      A     #i_TRS2_EXT_Inputs.Request_Stop; // IF External stop Request
      O     #s_TRS2_ST_PEC_Block; // OR PEC blockage
      O     #o_TRS2_ST_PPI_Err; // OR PPI error
      O     #s_TRS2_ST_LMS_ASI_Not_Pr; // OR LMS ASI not present
      O     #s_TRS2_ST_LMS_ASI_Error; // OR LMS ASI Error
      O     #s_TRS2_ST_LMS_Not_Health; // OR LMS not healthy
      O     #s_TRS2_ST_PEC_Missings; // OR PEC missing
      O     #s_TRS2_ST_LMS_Not_Auto; // OR in automatic mode
      O     #s_Req_Stop_TRS2; // OR request to stop TRS 2 due to error of VBS or SWS
      =     #s_TRS2_Req_Stop; // Request Stop

// Request Halt to the section
      A     #i_Ext_Req_Dis_Send;
      O     #s_Halt_TRS2_Gap_Not_Clr; // Halt TRS2 when the gap clear area is not clear and the divert section is not running
      O     #s_Halt_TRS2_Dir1;
      O     #s_Halt_TRS2_Dir2;
      O     #s_Halt_TRS2_Belt_NOK;
      O     #s_DecPoint_Wait_TRS2; // Settings at decision point are configured to halt the item in front of the vertibelt
      O     #i_TRS2_EXT_Inputs.Request_Halt; // IF External halt Request
      =     #s_TRS2_Req_Halt;

      CALL "FC_PLT_Clr_DB" (
           i_Enable_Clr             := #s_TRS2_ST_LMS_Not_Auto,
           i_DB_PLT_Num             := #t_DB_PLT_TRS2,
           i_DB_Event_Num           := #s_DB_Num_Event);

      CALL #s_TRS2_FB_EQP_Basic (
           i_ID_Section             := #i_TRS2_ID,
           i_Setting                := #i_TRS2_Setting.Basic,
           i_DB_PLT                 := #i_TRS2_DB_PLT,
           i_DB_PLT_DwnStr          := #i_TRS2_DB_PLT_Downstr,
           i_DB_Event               := "DB_Event_Section",
           i_CFG_Conveyor_Speed     := #i_TRS2_CFG_Conv_Speed,
           i_CFG_Run_Out_Distance   := #i_TRS2_CFG_Run_Out_Dist,
           i_CFG_Minimum_Gap        := #i_CFG_TRS2_Minimum_Gap,
           i_CFG_Add_Gap_Stop       := #i_CFG_TRS2_Add_Gap_Stop,
           i_CFG_Minimum_H2H        := #i_CFG_TRS2_Minimum_H2H,
           i_CFG_Add_H2H_Stop       := #i_CFG_TRS2_Add_H2H_Stop,
           i_CFG_Cascade_Delay_Time := 300,
           i_CFG_Strt_Up_T_E_Save   := "DB_Setting".common.Start_Up_Time_E_Save,
           i_CFG_Run_Out_E_Save     := "DB_Setting".common.Run_Out_Time_E_Save,
           i_CFG_Stop_T_E_Save      := "DB_Setting".common.Stop_Time_E_Save,
           i_CFG_Disbl_E_Save       := "DB_Setting".common.Disable_Energy_Saving,
           i_CFG_Slave_Mode         := FALSE,
           i_CFG_Del_Window_Codes   := FALSE,
           i_PPI_Displacement       := 0,
           i_Dwnstr_PLT_Pos         := #s_TRS2_Int_Prog.PEC_Offset,
           i_Available_IO           := #i_TRS2_Available_IO,
           i_Safety_OK              := #i_Safety_OK,
           i_CMD_Enable             := #i_CMD_Enable,
           i_CMD_Start              := #i_CMD_Start,
           i_Ext_Req_Stop           := #s_TRS2_Req_Stop,
           i_Ext_Req_Halt           := #s_TRS2_Req_Halt,
           i_Ext_Req_Dis_Send       := #i_TRS2_EXT_Inputs.Request_Disable_Send,
           i_Ext_Req_Rst_ESave      := #i_TRS2_EXT_Inputs.Request_Reset_EnergySave,
           i_OS_Direction_Change    := FALSE,
           o_External               := #o_TRS2_EXT_Outputs,
           o_Motor_Run              := #s_TRS2_Int_Prog.Motor_Run,
           o_ST_Items               := #o_TRS2_ST_Items,
           o_ST_Running             := #o_TRS2_ST_Running,
           o_ST_Started             := #o_TRS2_ST_Started,
           o_ST_Request_Halt        := #o_TRS2_ST_Req_Halt,
           o_ST_Request_Stop        := #o_TRS2_ST_Req_Stop,
           o_Ready_To_Restart       := #s_TRS2_Ready_Restart);

      CALL #s_TRS2_FB_TRK_Track (
           i_Trigger_Send_Stat      := #i_CMD_Send_Stat,
           i_CMD_Reset              := #i_CMD_Reset,
           i_DB_PLT                 := #i_TRS2_DB_PLT,
           i_Event_DB               := "DB_Event_Section",
           i_Position_PEC_Update    := #s_TRS2_Int_Prog.PEC_Offset,
           i_LPOS                   := #s_TRS2_Int_Prog.LPOS,
           i_Setting                := #i_TRS2_Setting.Tracking,
           i_CFG_Clear_Double_Data  := FALSE,
           i_Length_Dif_Accepted    := 0,
           i_CFG_Num_Missing_Error  := 3,
           i_CFG_Upd_Perf_WN_Level  := 80,
           i_CFG_Weighing_Factor    := 10,
           i_CFG_Default_Record     := #i_CFG_Default_Record,
           i_OS_Direction_Change    := FALSE,
           o_ST_PEC_Miss            := #s_TRS2_ST_PEC_Missings,
           o_ST_PEC_BadTrack        := #o_TRS2_ST_Bad_Update);

      CALL #s_TRS2_FB_HW_MTR_LMS (
           i_CMD_Send_Stat          := #i_CMD_Send_Stat,
           i_Event_DB               := "DB_Event_Section",
           i_Available_IO           := #i_TRS2_Available_IO,
           i_Quick_Stop             := FALSE,
           i_LMS_NotPrsnt           := #i_TRS2_IO_LMS_NotPrsnt,
           i_LMS_Error              := #i_TRS2_IO_LMS_Error,
           i_IO_LMS_Auto            := #i_TRS2_IO_LMS_Auto,
           i_IO_LMS_Healthy         := #i_TRS2_IO_LMS_Healthy,
           i_CMD_Reset              := #i_CMD_Reset,
           i_CMD_Req_Motor_Forward  := #s_TRS2_Int_Prog.Motor_Run,
           o_IO_MTR_Fwd             := #o_TRS2_IO_MTR_Fwd,
           o_IO_MTR_Rev             := #o_TRS2_IO_MTR_Rev,
           o_IO_MTR_Dis_Quick_Stop  := #o_TRS2_IO_Disable_QS,
           o_ST_ASI_NotPrsnt        := #s_TRS2_ST_LMS_ASI_Not_Pr,
           o_ST_ASI_Err             := #s_TRS2_ST_LMS_ASI_Error,
           o_ST_LMS_Not_Auto        := #s_TRS2_ST_LMS_Not_Auto,
           o_ST_LMS_Not_Hthy        := #s_TRS2_ST_LMS_Not_Health);

      CALL #s_TRS2_Window_Generator (
           i_DB_PLT_Most_DwnStr     := #i_TRS2_DB_PLT,
           i_DB_PLT_Most_UpStr      := #i_TRS2_DB_PLT,
           i_DB_Reservation         := #i_DB_Res_TRS2,
           i_DB_Event               := "DB_Event_Zone",
           i_CFG_Window_Length      := #s_Calc_H2H_Length_VBS1,
           i_CFG_In_Flow_Function   := FALSE,
           i_Section_Run_Reverse    := FALSE);

      CALL #s_FB_DAT_TRS2 (
           i_ID_Section             := #i_TRS2_ID,
           i_DB_Event               := "DB_Event_Section",
           i_PLC_FIFO_DB            := "DB_Send_FIFO",
           i_PLC_Log_FIFO_DB        := "DB_LOG_Event_FIFO",
           i_Degraded_Mode          := "M_Comm_Degraded",
           i_CFG_BPI_Log_Level      := "DB_Setting".common.External_Log_Level,
           i_CFG_PLC_Log_Level      := "DB_Setting".common.Internal_Log_Level,
           i_CFG_PLC_Log_SAC_Mesgs  := FALSE,
           i_CFG_PLC_LOG_BPI_Stat   := FALSE);

NETWORK
TITLE =UA: Right sorter section (TRS3)

      NOP   0;
// Induct from section upstream of TRS3 onto TRS3 is only used when flow A is active
      A     #s_Flow_A;
      JCN   UA01;

      CALL #s_TRS3_FB_Induct (
           i_Setting                := #i_Setting.Induct_Upstr_TRS3_Sett,
           i_DB_PLT                 := #i_TRS3_Ups_Induct_DB_PLT,
           i_DB_PLT_Merge           := #i_TRS3_DB_PLT,
           i_DB_Reservation         := #i_DB_Res_TRS3,
           i_DB_Event               := "DB_Event_Zone",
           i_CFG_PEC_Offset         := #s_TRS3_Int_Prog.PEC_Offset,
           i_CFG_Search_Window      := 0,
           i_CFG_Gap_Length         := 20,
           i_CFG_Induct_Number_FWD  := 2,
           i_CFG_Run_Out_Dist_Gap   := #i_TRS3_Ups_Run_Out_Dist);

// When using the induct block connect the induct PLT DB inbetween TRS3 and it's upstream section
      OPN   #i_TRS3_DB_PLT;
      L     0; //#s_Upst_TRS3_IND_DB_PLT
      T     DBW    6;

      OPN   #i_TRS3_DB_PLT_Upstr;
      L     #s_Upst_TRS3_IND_DB_PLT;
      T     DBW    8;

      OPN   #i_TRS3_Ups_Induct_DB_PLT;
      L     #s_TRS3_DB_PLT_Upstream;
      T     DBW    6;
      L     #t_DB_PLT_TRS3;
      T     DBW    8;
      JU    UA02;

// When not using the induct block connect TRS3 direct to it's upstream section.
UA01: OPN   #i_TRS3_DB_PLT;
      L     #s_TRS3_DB_PLT_Upstream;
      T     DBW    6;

      OPN   #i_TRS3_DB_PLT_Upstr;
      L     #t_DB_PLT_TRS3;
      T     DBW    8;

UA02: NOP   0;

      CALL "FC_Calc_H2H_Distance" (
           i_CFG_Conveyor_Speed     := #i_TRS3_CFG_Conv_Speed,
           i_CFG_Capacity           := 1200,
           i_CFG_Minimum_Capacity   := 1200,
           i_CFG_Maximum_Capacity   := 1200,
           o_H2H_Length             := #s_Calc_H2H_Length_VBS2,
           o_Current_Capacity       := #o_Capacity_VBS2,
           o_ST_Capacity_2Low       := #t_Not_Used_Bool,
           o_ST_Capacity_2High      := #t_Not_Used_Bool,
           o_ST_CalcH2H_Disable     := #t_Not_Used_Bool);

      CALL #s_TRS3_FB_EQP_PEC (
           i_Setting                := #i_TRS3_Setting.PEC_1D,
           i_DB_PLT                 := #i_TRS3_DB_PLT,
           i_DB_Event               := "DB_Event_Section",
           i_Dwnstr_PLT_Pos         := 0,
           i_CFG_Blockage_Length    := 300,
           i_CFG_Delay_On_Filter    := 0,
           i_CFG_Delay_Off_Filter   := 20,
           i_CFG_Min_Product_Length := 0,
           i_CFG_Preset_PEC_Latch   := #s_TRS3_ST_LMS_Not_Auto,
           i_CFG_Track_Present      := TRUE,
           i_CFG_Reset_Block_PEC_Oc := FALSE,
           i_IO_NOT_PEC             := #i_TRS3_IO_NOT_PEC,
           i_Eqp_Available_IO       := #i_TRS3_Available_IO,
           i_CMD_Reset              := #i_CMD_Reset,
           o_LPOS                   := #s_TRS3_Int_Prog.LPOS,
           o_PEC_Position           := #s_TRS3_Int_Prog.PEC_Offset,
           o_ST_PEC_Blk             := #s_TRS3_ST_PEC_Block);

      CALL #s_TRS3_FB_EQP_PPI (
           i_CFG_PPI_Resolution     := 50,
           i_CFG_Time_Out_Error     := 300,
           i_DB_PLT                 := #i_TRS3_DB_PLT,
           i_IO_PPI                 := #i_TRS3_IO_PPI,
           i_CMD_Reset              := #i_CMD_Reset,
           o_PPI_Displacement_mm    := #s_TRS3_Int_Prog.PPI_Displacement,
           o_ST_PPI_Err             := #o_TRS3_ST_PPI_Err);

// Request stop for basic equipment
      A     #s_VBS2_ST_Not_Automatic;
      O     #s_SWS_VBS2_Gap_NotClr;
      O     #s_SWS2_ST_Move_Time_Out;
      O     #s_VBS2_ST_Not_Healthy;
      O     #s_VBS2_ST_ASI_Not_Prsnt;
      O     #s_VBS2_ST_ASI_Error;
      O     #s_SWS2_ST_ASI_Not_Presnt;
      O     #s_SWS2_ST_ASI_Error;
      O     #s_SWS2_ST_Err_PS_Double;
      O     #s_TRS1_ST_PEC_Block_1;
      =     #s_Req_Stop_TRS3;

      A     #i_TRS3_EXT_Inputs.Request_Stop; // IF External stop Request
      O     #s_TRS3_ST_PEC_Block; // OR PEC blockage
      O     #o_TRS3_ST_PPI_Err; // OR PPI error
      O     #s_TRS3_ST_LMS_ASI_Not_Pr; // OR LMS ASI not present
      O     #s_TRS3_ST_LMS_ASI_Error; // OR LMS ASI Error
      O     #s_TRS3_ST_LMS_Not_Health; // OR LMS not healthy
      O     #s_TRS3_ST_PEC_Missings; // OR PEC missing
      O     #s_TRS3_ST_LMS_Not_Auto; // OR in automatic mode
      O     #s_Req_Stop_TRS3;
      =     #s_TRS3_Req_Stop; // Request Stop

// Request Halt to the section
      A     #i_Ext_Req_Dis_Send;
      O     #s_Halt_TRS3_Gap_Not_CLR; // Halt TRS3 when the gap clear area is not clear and the divert section is not running
      O     #s_Halt_TRS3_Dir1;
      O     #s_Halt_TRS3_Dir2;
      O     #s_Halt_TRS3_Belt_NOK;
      O     #s_DecPoint_Wait_TRS3; // Settings at decision point are configured to halt the item in front of the vertibelt
      O     #i_TRS3_EXT_Inputs.Request_Halt; // IF External halt Request
      =     #s_TRS3_Req_Halt;

      CALL "FC_PLT_Clr_DB" (
           i_Enable_Clr             := #s_TRS3_ST_LMS_Not_Auto,
           i_DB_PLT_Num             := #t_DB_PLT_TRS3,
           i_DB_Event_Num           := #s_DB_Num_Event);

      CALL #s_TRS3_FB_EQP_Basic (
           i_ID_Section             := #i_TRS3_ID,
           i_Setting                := #i_TRS3_Setting.Basic,
           i_DB_PLT                 := #i_TRS3_DB_PLT,
           i_DB_PLT_DwnStr          := #i_TRS3_DB_PLT_Downstream,
           i_DB_Event               := "DB_Event_Section",
           i_CFG_Conveyor_Speed     := #i_TRS3_CFG_Conv_Speed,
           i_CFG_Run_Out_Distance   := #i_TRS3_CFG_Run_Out_Dist,
           i_CFG_Minimum_Gap        := #i_CFG_TRS3_Minimum_Gap,
           i_CFG_Add_Gap_Stop       := #i_CFG_TRS3_Add_Gap_Stop,
           i_CFG_Minimum_H2H        := #i_CFG_TRS3_Minimum_H2H,
           i_CFG_Add_H2H_Stop       := #i_CFG_TRS3_Add_H2H_Stop,
           i_CFG_Cascade_Delay_Time := 300,
           i_CFG_Strt_Up_T_E_Save   := "DB_Setting".common.Start_Up_Time_E_Save,
           i_CFG_Run_Out_E_Save     := "DB_Setting".common.Run_Out_Time_E_Save,
           i_CFG_Stop_T_E_Save      := "DB_Setting".common.Stop_Time_E_Save,
           i_CFG_Disbl_E_Save       := "DB_Setting".common.Disable_Energy_Saving,
           i_CFG_Slave_Mode         := FALSE,
           i_CFG_Del_Window_Codes   := FALSE,
           i_PPI_Displacement       := 0,
           i_Dwnstr_PLT_Pos         := #s_TRS3_Int_Prog.PEC_Offset,
           i_Available_IO           := #i_TRS3_Available_IO,
           i_Safety_OK              := #i_Safety_OK,
           i_CMD_Enable             := #i_CMD_Enable,
           i_CMD_Start              := #i_CMD_Start,
           i_Ext_Req_Stop           := #s_TRS3_Req_Stop,
           i_Ext_Req_Halt           := #s_TRS3_Req_Halt,
           i_Ext_Req_Dis_Send       := #i_TRS3_EXT_Inputs.Request_Disable_Send,
           i_Ext_Req_Rst_ESave      := #i_TRS3_EXT_Inputs.Request_Reset_EnergySave,
           i_OS_Direction_Change    := FALSE,
           o_External               := #o_TRS3_EXT_Outputs,
           o_Motor_Run              := #s_TRS3_Int_Prog.Motor_Run,
           o_ST_Items               := #o_TRS3_ST_Items,
           o_ST_Running             := #o_TRS3_ST_Running,
           o_ST_Started             := #o_TRS3_ST_Started,
           o_ST_Request_Halt        := #o_TRS3_ST_Req_Halt,
           o_ST_Request_Stop        := #o_TRS3_ST_Req_Stop,
           o_Ready_To_Restart       := #s_TRS3_Ready_Restart);

      CALL #s_TRS3_FB_TRK_Track (
           i_Trigger_Send_Stat      := #i_CMD_Send_Stat,
           i_CMD_Reset              := #i_CMD_Reset,
           i_DB_PLT                 := #i_TRS3_DB_PLT,
           i_Event_DB               := "DB_Event_Section",
           i_Position_PEC_Update    := #s_TRS3_Int_Prog.PEC_Offset,
           i_LPOS                   := #s_TRS3_Int_Prog.LPOS,
           i_Setting                := #i_TRS3_Setting.Tracking,
           i_CFG_Clear_Double_Data  := FALSE,
           i_Length_Dif_Accepted    := 0,
           i_CFG_Num_Missing_Error  := 3,
           i_CFG_Upd_Perf_WN_Level  := 80,
           i_CFG_Weighing_Factor    := 10,
           i_CFG_Default_Record     := #i_CFG_Default_Record,
           i_OS_Direction_Change    := FALSE,
           o_ST_PEC_Miss            := #s_TRS3_ST_PEC_Missings,
           o_ST_PEC_BadTrack        := #o_TRS3_ST_Bad_Update);

      CALL #s_TRS3_FB_HW_MTR_LMS (
           i_CMD_Send_Stat          := #i_CMD_Send_Stat,
           i_Event_DB               := "DB_Event_Section",
           i_Available_IO           := #i_TRS3_Available_IO,
           i_Quick_Stop             := FALSE,
           i_LMS_NotPrsnt           := #i_TRS3_IO_LMS_NotPrsnt,
           i_LMS_Error              := #i_TRS3_IO_LMS_Error,
           i_IO_LMS_Auto            := #i_TRS3_IO_LMS_Auto,
           i_IO_LMS_Healthy         := #i_TRS3_IO_LMS_Healthy,
           i_CMD_Reset              := #i_CMD_Reset,
           i_CMD_Req_Motor_Forward  := #s_TRS3_Int_Prog.Motor_Run,
           o_IO_MTR_Fwd             := #o_TRS3_IO_MTR_Fwd,
           o_IO_MTR_Rev             := #o_TRS3_IO_MTR_Rev,
           o_IO_MTR_Dis_Quick_Stop  := #o_TRS3_IO_Disable_QS,
           o_ST_ASI_NotPrsnt        := #s_TRS3_ST_LMS_ASI_Not_Pr,
           o_ST_ASI_Err             := #s_TRS3_ST_LMS_ASI_Error,
           o_ST_LMS_Not_Auto        := #s_TRS3_ST_LMS_Not_Auto,
           o_ST_LMS_Not_Hthy        := #s_TRS3_ST_LMS_Not_Health);

      CALL #s_TRS3_Window_Generator (
           i_DB_PLT_Most_DwnStr     := #i_TRS3_DB_PLT,
           i_DB_PLT_Most_UpStr      := #i_TRS3_DB_PLT,
           i_DB_Reservation         := #i_DB_Res_TRS3,
           i_DB_Event               := "DB_Event_Zone",
           i_CFG_Window_Length      := #s_Calc_H2H_Length_VBS2,
           i_CFG_In_Flow_Function   := FALSE,
           i_Section_Run_Reverse    := FALSE);

      CALL #s_FB_DAT_TRS3 (
           i_ID_Section             := #i_TRS3_ID,
           i_DB_Event               := "DB_Event_Section",
           i_PLC_FIFO_DB            := "DB_Send_FIFO",
           i_PLC_Log_FIFO_DB        := "DB_LOG_Event_FIFO",
           i_Degraded_Mode          := "M_Comm_Degraded",
           i_CFG_BPI_Log_Level      := "DB_Setting".common.External_Log_Level,
           i_CFG_PLC_Log_Level      := "DB_Setting".common.Internal_Log_Level,
           i_CFG_PLC_Log_SAC_Mesgs  := FALSE,
           i_CFG_PLC_LOG_BPI_Stat   := FALSE);

NETWORK
TITLE =VA: Data Layer of VBZ
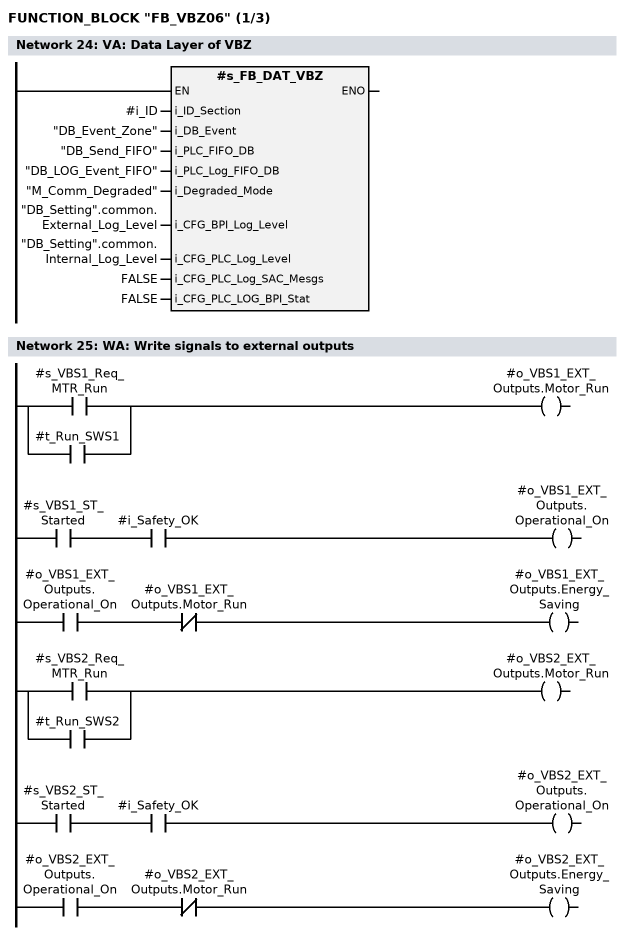

      CALL #s_FB_DAT_VBZ (
           i_ID_Section             := #i_ID,
           i_DB_Event               := "DB_Event_Zone",
           i_PLC_FIFO_DB            := "DB_Send_FIFO",
           i_PLC_Log_FIFO_DB        := "DB_LOG_Event_FIFO",
           i_Degraded_Mode          := "M_Comm_Degraded",
           i_CFG_BPI_Log_Level      := "DB_Setting".common.External_Log_Level,
           i_CFG_PLC_Log_Level      := "DB_Setting".common.Internal_Log_Level,
           i_CFG_PLC_Log_SAC_Mesgs  := FALSE,
           i_CFG_PLC_LOG_BPI_Stat   := FALSE);

NETWORK
TITLE =WA: Write signals to external outputs

      NOP   0;
// Signals for VBS 1
      A     #s_VBS1_Req_MTR_Run;
      O     #t_Run_SWS1;
      =     #o_VBS1_EXT_Outputs.Motor_Run;

      A     #s_VBS1_ST_Started;
      A     #i_Safety_OK;
      =     #o_VBS1_EXT_Outputs.Operational_On;

      A     #o_VBS1_EXT_Outputs.Operational_On;
      AN    #o_VBS1_EXT_Outputs.Motor_Run;
      =     #o_VBS1_EXT_Outputs.Energy_Saving;

// Signals for VBS 2
      A     #s_VBS2_Req_MTR_Run;
      O     #t_Run_SWS2;
      =     #o_VBS2_EXT_Outputs.Motor_Run;

      A     #s_VBS2_ST_Started;
      A     #i_Safety_OK;
      =     #o_VBS2_EXT_Outputs.Operational_On;

      A     #o_VBS2_EXT_Outputs.Operational_On;
      AN    #o_VBS2_EXT_Outputs.Motor_Run;
      =     #o_VBS2_EXT_Outputs.Energy_Saving;
NETWORK
TITLE =XA: Write zone status
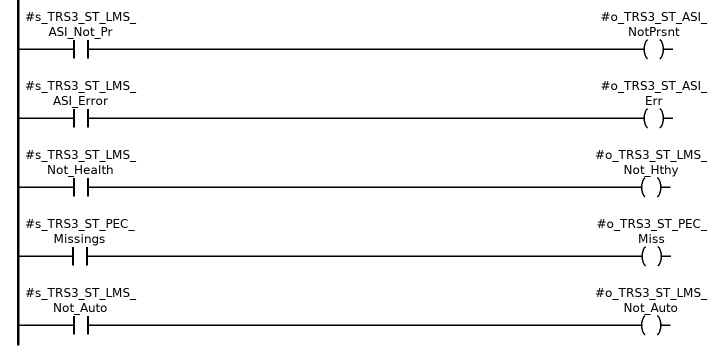

      A     #s_Flow_Straight;
      =     #o_ST_Fixed_Straight;

      A     #s_Flow_A;
      =     #o_ST_Fixed_Flow_A;

      A     #s_Flow_B;
      =     #o_ST_Fixed_Flow_B;

      A     #s_VBS1_ST_Started;
      AN    #s_VBS1_ST_Not_Automatic;
      AN    #s_VBS1_ST_Not_Healthy;
      AN    #s_VBS1_ST_ASI_Not_Prsnt;
      AN    #s_VBS1_ST_ASI_Error;
      =     #o_VBS1_ST_Started;

      A     #s_VBS2_ST_Started;
      AN    #s_VBS2_ST_Not_Automatic;
      AN    #s_VBS2_ST_Not_Healthy;
      AN    #s_VBS2_ST_ASI_Not_Prsnt;
      AN    #s_VBS2_ST_ASI_Error;
      =     #o_VBS2_ST_Started;

// Copy section statusses to outputs

      A     #s_VBS1_ST_ASI_Not_Prsnt;
      =     #o_VBS1_ST_ASI_NotPrsnt;

      A     #s_VBS1_ST_ASI_Error;
      =     #o_VBS1_ST_ASI_Err;

      A     #s_VBS1_ST_Not_Automatic;
      =     #o_VBS1_ST_LMS_Not_Auto;

      A     #s_VBS1_ST_Not_Healthy;
      =     #o_VBS1_ST_LMS_Not_Hthy;

      A     #s_SWS1_ST_ASI_Not_Presnt;
      =     #o_SWS1_ST_ASI_NotPrsnt;

      A     #s_SWS1_ST_ASI_Error;
      =     #o_SWS1_ST_ASI_Error;

      A     #s_SWS1_ST_Not_Automatic;
      =     #o_SWS1_ST_Not_Automatic;

      A     #s_SWS1_ST_Not_Healthy;
      =     #o_SWS1_ST_Not_Healthy;

      A     #s_SWS1_ST_Move_Time_Out;
      =     #o_SWS1_ST_Move_Time_Out;

      A     #s_SWS1_ST_Err_PS_Double;
      =     #o_SWS1_ST_Err_PS_Double;

      A     #s_VBS2_ST_ASI_Not_Prsnt;
      =     #o_VBS2_ST_ASI_NotPrsnt;

      A     #s_VBS2_ST_ASI_Error;
      =     #o_VBS2_ST_ASI_Err;

      A     #s_VBS2_ST_Not_Automatic;
      =     #o_VBS2_ST_LMS_Not_Auto;

      A     #s_VBS2_ST_Not_Healthy;
      =     #o_VBS2_ST_LMS_Not_Hthy;

      A     #s_SWS2_ST_ASI_Not_Presnt;
      =     #o_SWS2_ST_ASI_NotPrsnt;

      A     #s_SWS2_ST_ASI_Error;
      =     #o_SWS2_ST_ASI_Error;

      A     #s_SWS2_ST_Not_Automatic;
      =     #o_SWS2_ST_Not_Automatic;

      A     #s_SWS2_ST_Not_Healthy;
      =     #o_SWS2_ST_Not_Healthy;

      A     #s_SWS2_ST_Move_Time_Out;
      =     #o_SWS2_ST_Move_Time_Out;

      A     #s_SWS2_ST_Err_PS_Double;
      =     #o_SWS2_ST_Err_PS_Double;

      A     #s_TRS1_ST_PEC_Block_1;
      =     #o_TRS1_ST_PEC_Blk;

      A     #s_TRS1_ST_PEC_Block_2;
      =     #o_TRS1_ST_PEC2_Blk;

      A     #s_TRS1_ST_LMS_ASI_Not_Pr;
      =     #o_TRS1_ST_ASI_NotPrsnt;

      A     #s_TRS1_ST_LMS_ASI_Error;
      =     #o_TRS1_ST_ASI_Err;

      A     #s_TRS1_ST_LMS_Not_Health;
      =     #o_TRS1_ST_LMS_Not_Hthy;

      A     #s_TRS1_ST_PEC_Missings;
      =     #o_TRS1_ST_PEC_Miss;

      A     #s_TRS1_ST_LMS_Not_Auto;
      =     #o_TRS1_ST_LMS_Not_Auto;

      A     #s_TRS2_ST_PEC_Block;
      =     #o_TRS2_ST_PEC_Blk;

      A     #s_TRS2_ST_LMS_ASI_Not_Pr;
      =     #o_TRS2_ST_ASI_NotPrsnt;

      A     #s_TRS2_ST_LMS_ASI_Error;
      =     #o_TRS2_ST_ASI_Err;

      A     #s_TRS2_ST_LMS_Not_Health;
      =     #o_TRS2_ST_LMS_Not_Hthy;

      A     #s_TRS2_ST_PEC_Missings;
      =     #o_TRS2_ST_PEC_Miss;

      A     #s_TRS2_ST_LMS_Not_Auto;
      =     #o_TRS2_ST_LMS_Not_Auto;

      A     #s_TRS3_ST_PEC_Block;
      =     #o_TRS3_ST_PEC_Blk;

      A     #s_TRS3_ST_LMS_ASI_Not_Pr;
      =     #o_TRS3_ST_ASI_NotPrsnt;

      A     #s_TRS3_ST_LMS_ASI_Error;
      =     #o_TRS3_ST_ASI_Err;

      A     #s_TRS3_ST_LMS_Not_Health;
      =     #o_TRS3_ST_LMS_Not_Hthy;

      A     #s_TRS3_ST_PEC_Missings;
      =     #o_TRS3_ST_PEC_Miss;

      A     #s_TRS3_ST_LMS_Not_Auto;
      =     #o_TRS3_ST_LMS_Not_Auto;

NETWORK
TITLE =YA: Write zone status request signals
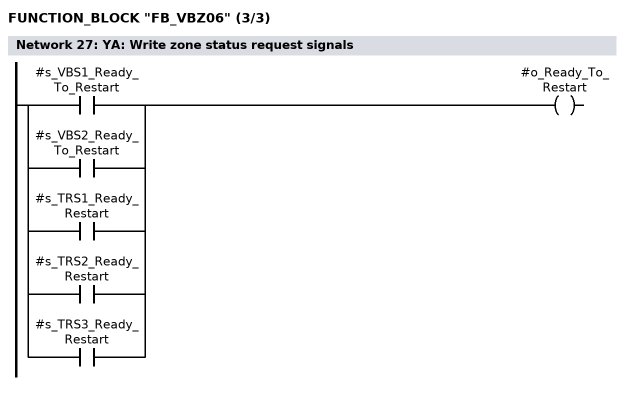

      O     #s_VBS1_Ready_To_Restart;
      O     #s_VBS2_Ready_To_Restart;
      O     #s_TRS1_Ready_Restart;
      O     #s_TRS2_Ready_Restart;
      O     #s_TRS3_Ready_Restart;
      =     #o_Ready_To_Restart;
END_FUNCTION_BLOCK

